KUKA KRL program: chk_w6_rps2_opn.src

&ACCESS RVO8
&COMMENT Check RPS AXOR Z2 OPEN
DEF chk_w6_rps2_opn( )

; Check rps axor OPEN Z2.1
;//---- Start User-------

$TIMER[10] = 0
$TIMER_STOP[10] = FALSE

WAIT FOR ($IN[495])
WAIT FOR (NOT $IN[496])

$TIMER_STOP[10] = TRUE
$TIMER[10] = 0

;//---- End User---------
END
